FUNCTION RESET_ZONA_OUTPUT : ZONA_INPUT

VAR_INPUT
	INPUT : ZONA_OUTPUT;
END_VAR

VAR_OUTPUT
	OUTPUT : ZONA_OUTPUT;
END_VAR

INPUT.LIBERO := FALSE;
INPUT.TRIGGER := FALSE;
OUTPUT := INPUT;

END_FUNCTION

(* stored: Version 1.1.0.1, ProductVersion 3.1.4024.12
   POU RESET_ZONA_OUTPUT: Id {897f9b47-f23e-4337-9ae0-eb90d8fef53f}, SpecialFunc None *)
